// TwinCAT 3 PLC project PLC
// Title: TcMeasurementBridge
// Company: Roald
// Author: Roald
// ProjectVersion: 0.1.0
// Description: Function blocks to communicate with EL3356 measurement bridge to measure resistor bridges of load cells for example.
// ProgramVersion: 3.1.4023.0
// libraries:
//   Tc2_Standard, * (Beckhoff Automation GmbH)
//   Tc2_System, * (Beckhoff Automation GmbH)
//   Tc3_Module, * (Beckhoff Automation GmbH)
//   TcCoE, * (Roald)
//   TcError, * (Roald)
//   TcLog, * (Benedikt Geisler)
//   TcUnits, * (Roald)
// project tree:
//   LoadCell/ EL3356_CoE.TcGVL, LoadCell.TcPOU, LoadCellParameterizationSteps.TcDUT, ResistorMeasurementBridgeSettings.TcDUT
//   / PlcTask.TcTTO (not stored)

// ---- LoadCell/LoadCellParameterizationSteps.TcDUT
{attribute 'qualified_only'}
{attribute 'strict'}
{attribute 'to_string'}
TYPE LoadCellParameterizationSteps : (
    resetToFactorySettings := 0,
    setRatedOutput,
    setNominalLoad,
    setNominalOffset,
    setScalingFactor,
    Done
);
END_TYPE

// ---- LoadCell/ResistorMeasurementBridgeSettings.TcDUT
TYPE ResistorMeasurementBridgeSettings : STRUCT
    ratedOutput : REAL; // Nominal characteristic value of the sensor element in mV/V
    nominalLoad : REAL; // Nominal load of the force transducer/load cell/etc. (e.g. in kg, N etc,)
    nominalOffset : REAL; // Zero point offset in mV/V
    scaleFactor : REAL; // This factor can be used to re-scale the process data. In order to change the display from kg to g, for example, the factor 1000 can be entered here.
END_STRUCT
END_TYPE

// ---- LoadCell/EL3356_CoE.TcGVL
{attribute 'qualified_only'}
VAR_GLOBAL CONSTANT
    parameterReset : DWORD := 16#64616F6C;
    parameterResetIndex : ProcessDataObjectIndex := (index:=16#1011, subIndex:=1);
    rmbRatedOutput : ProcessDataObjectIndex := (index:=16#8000, subIndex:=16#23);
    rmbNominalLoad : ProcessDataObjectIndex := (index:=16#8000, subIndex:=16#24);
    rmbNominalOffset : ProcessDataObjectIndex := (index:=16#8000, subIndex:=16#25);
    rmbScaling : ProcessDataObjectIndex := (index:=16#8000, subIndex:=16#27);
    {attribute 'analysis' := '-33'} // parameter is used, but not seen by the compiler
    sauter300Settings : ResistorMeasurementBridgeSettings := (
        nominalLoad:=300,
        nominalOffset:=0,
        ratedOutput:=2,
        scaleFactor:=1000
    );
END_VAR

// ---- LoadCell/LoadCell.TcPOU
FUNCTION_BLOCK LoadCell
VAR_INPUT
    inLoad AT %I* : DINT; // gram
END_VAR
VAR
    _amsAddress : AmsNetAddress;
    _settings : ResistorMeasurementBridgeSettings;

    _parameterizeSteps : LoadCellParameterizationSteps;
    _initialized : BOOL;
    {attribute 'analysis' := '-33'} // parameter is used, but not seen by the compiler
    _emptyAddress : AmsNetAddress;
    _coeWrite : CoeWriterEx(amsNetAddress:=_emptyAddress);
    _load : Kilogram;

    _logger : TcLog;
END_VAR

// Needs to be tested again, has been rewritten
IF NOT _initialized THEN
    Initialize();
ELSE
    _load := TO_LREAL(inLoad) / _settings.scaleFactor;
END_IF

{attribute 'hide'}
METHOD FB_init : BOOL
VAR_INPUT
    bInitRetains : BOOL; // if TRUE, the retain variables are initialized (warm start / cold start)
    bInCopyCode :
        BOOL; // if TRUE, the instance afterwards gets moved into the copy code (online change)
    amsAddress : AmsNetAddress;
    settings : ResistorMeasurementBridgeSettings;
END_VAR
THIS^._amsAddress := amsAddress;
THIS^._settings := settings;
_coeWrite.FB_init(bInitRetains:=bInitRetains, bInCopyCode:=bInCopyCode, amsNetAddress:=amsAddress);
END_METHOD

METHOD PRIVATE Initialize
IF NOT _coeWrite.bBusy THEN
    _coeWrite(bExecute:=FALSE);
END_IF

_logger.OnCondition(NOT _coeWrite.bBusy)
    .AppendString('Load cell reset at AMSID: ')
    .AppendAny(_coeWrite._amsNetAddress.netId)
    .AppendString(':')
    .AppendAny(_coeWrite._amsNetAddress.port).Debug('');
_logger.OnCondition(_coeWrite.bError)
    .AppendString('Failed to reset load cell reset to factory settings. Error:')
    .AppendAny(_coeWrite.eAdsError)
    .AppendString(': ')
    .AppendString(AdsErrorCodeDescription(_coeWrite.eAdsError)).Error('');

CASE _parameterizeSteps OF
    LoadCellParameterizationSteps.resetToFactorySettings:
        _coeWrite(
            index:=EL3356_CoE.parameterResetIndex,
            pSrcBuf:=ADR(EL3356_CoE.parameterReset),
            cbBufLen:=SIZEOF(EL3356_CoE.parameterReset),
            bExecute:=TRUE,
        );
        IF NOT _coeWrite.bBusy AND NOT _coeWrite.bError THEN
            _parameterizeSteps := LoadCellParameterizationSteps.setRatedOutput;
        END_IF
    LoadCellParameterizationSteps.setRatedOutput:
        _coeWrite(
            index:=EL3356_CoE.rmbRatedOutput,
            pSrcBuf:=ADR(_settings.ratedOutput),
            cbBufLen:=SIZEOF(_settings.ratedOutput),
            bExecute:=TRUE,
        );
        IF NOT _coeWrite.bBusy THEN
            _parameterizeSteps := LoadCellParameterizationSteps.setNominalLoad;
        END_IF
    LoadCellParameterizationSteps.setNominalLoad:
        _coeWrite(
            index:=EL3356_CoE.rmbNominalLoad,
            pSrcBuf:=ADR(_settings.nominalLoad),
            cbBufLen:=SIZEOF(_settings.nominalLoad),
            bExecute:=TRUE,
        );
        IF NOT _coeWrite.bBusy THEN
            _parameterizeSteps := LoadCellParameterizationSteps.setNominalOffset;
        END_IF
    LoadCellParameterizationSteps.setNominalOffset:
        _coeWrite(
            index:=EL3356_CoE.rmbNominalOffset,
            pSrcBuf:=ADR(_settings.nominalOffset),
            cbBufLen:=SIZEOF(_settings.nominalOffset),
            bExecute:=TRUE,
        );
        IF NOT _coeWrite.bBusy THEN
            _parameterizeSteps := LoadCellParameterizationSteps.setScalingFactor;
        END_IF
    LoadCellParameterizationSteps.setScalingFactor:
        _coeWrite(
            index:=EL3356_CoE.rmbScaling,
            pSrcBuf:=ADR(_settings.scaleFactor),
            cbBufLen:=SIZEOF(_settings.scaleFactor),
            bExecute:=TRUE,
        );
        IF NOT _coeWrite.bBusy THEN
            _parameterizeSteps := LoadCellParameterizationSteps.Done;
        END_IF
    LoadCellParameterizationSteps.Done:
        _initialized := TRUE;
END_CASE
END_METHOD

END_FUNCTION_BLOCK
